{region '#Template'}
	{attribute 'Version' := '5.0.1.0'}
	{attribute 'Tags' := '"LCID": "1031", "Text": "Universal, Motor, Aggregate"'}
	{attribute 'Tags' := '"LCID": "1033", "Text": "Universal, Motor, Aggregate"'}
	{attribute 'Using' := '"Type": "Template", "URI": "EC_ID"'}
	{attribute 'Using' := '"Type": "Template", "URI": "BA2_Param"'}
	{attribute 'Description' := '"LCID": "1031", "Text": "Motor modulierend mit Regler"'}
	{attribute 'Description' := '"LCID": "1033", "Text": "Motor modulating with controller"'}
{endregion}		
FUNCTION_BLOCK FB_BA_MotCtl EXTENDS FB_BA_View
VAR_INPUT
	fIn				: REAL;	// Istwert Regler // Actual value controller	
	stCmd			: ST_BA_Mdlt;
END_VAR
VAR_OUTPUT
	bCmd			: BOOL;
	fMdlt			: REAL;
	bDst			: BOOL;
	eActivePrio		: E_BA_Priority;
END_VAR

VAR_INPUT CONSTANT
	Dst				: FB_BA_BI_Raw;
	Cmd				: FB_BA_BO_Raw;								 
	Mdlt			: FB_BA_AO_Raw;							
	Sp				: FB_BA_AV_Op;		 
	Ctrl			: FB_BA_Loop;		
	PlantLock		: FB_BA_PlantLock;														
END_VAR
VAR
	bPrioSfty					: BOOL;
	bPrioCrit					: BOOL;	
	
	PrioSwiVal					: FB_BA_PrioSwi_UDI04;	

	MuxCmd						: FB_BA_MMUX_B04;
	MuxMdlt						: FB_BA_MMUX_R04;
	fMax						: REAL;
	fMin						: REAL;		
END_VAR
VAR // added by the converter: edge detectors and wires of the graphical bodies
    _w1, _w2 : ANY;
END_VAR

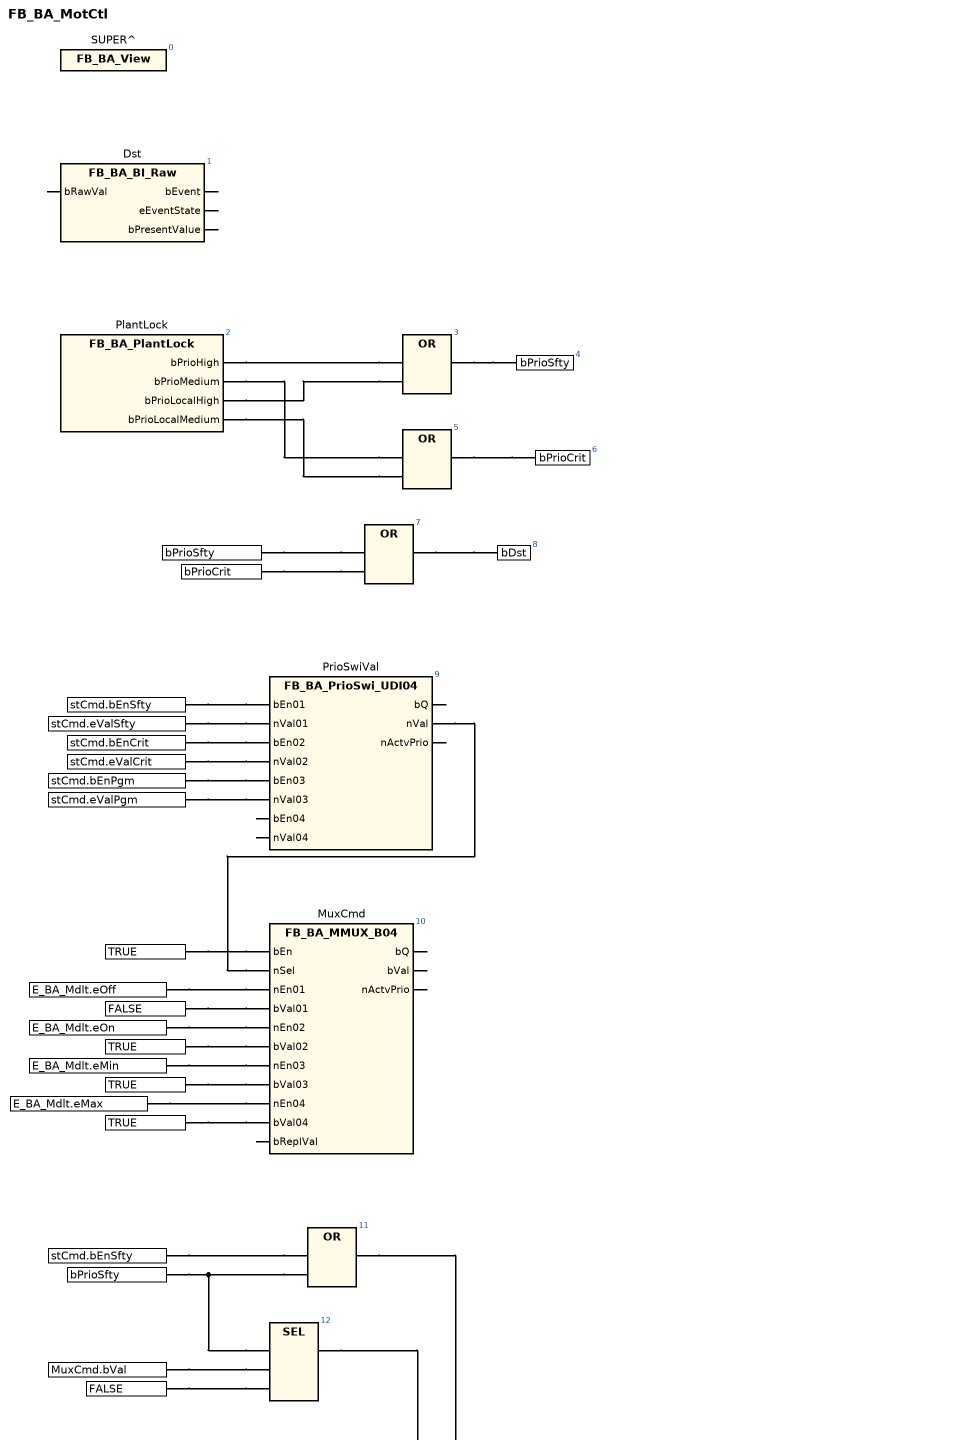
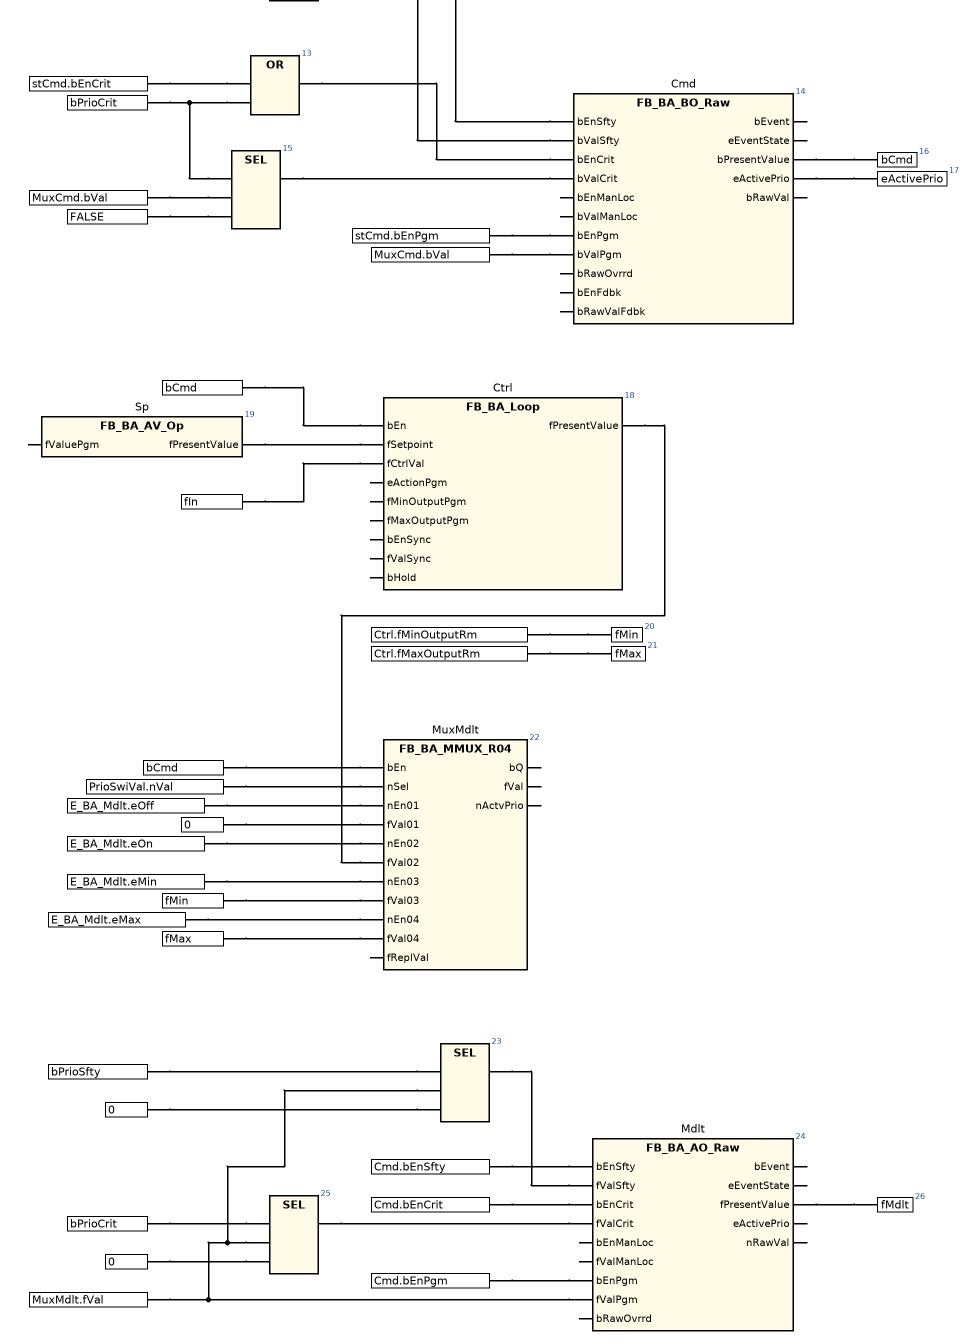
SUPER^(); // FB_BA_View
Dst(); // FB_BA_BI_Raw
PlantLock(); // FB_BA_PlantLock
bPrioSfty := PlantLock.bPrioHigh OR PlantLock.bPrioLocalHigh;
bPrioCrit := PlantLock.bPrioMedium OR PlantLock.bPrioLocalMedium;
bDst := bPrioSfty OR bPrioCrit;
PrioSwiVal(
    bEn01 := stCmd.bEnSfty,
    nVal01 := stCmd.eValSfty,
    bEn02 := stCmd.bEnCrit,
    nVal02 := stCmd.eValCrit,
    bEn03 := stCmd.bEnPgm,
    nVal03 := stCmd.eValPgm); // FB_BA_PrioSwi_UDI04
MuxCmd(
    bEn := TRUE,
    nSel := PrioSwiVal.nVal,
    nEn01 := E_BA_Mdlt.eOff,
    bVal01 := FALSE,
    nEn02 := E_BA_Mdlt.eOn,
    bVal02 := TRUE,
    nEn03 := E_BA_Mdlt.eMin,
    bVal03 := TRUE,
    nEn04 := E_BA_Mdlt.eMax,
    bVal04 := TRUE); // FB_BA_MMUX_B04
Cmd(
    bEnSfty := stCmd.bEnSfty OR bPrioSfty,
    bValSfty := SEL(bPrioSfty, MuxCmd.bVal, FALSE),
    bEnCrit := stCmd.bEnCrit OR bPrioCrit,
    bValCrit := _w1,
    bEnPgm := stCmd.bEnPgm,
    bValPgm := MuxCmd.bVal); // FB_BA_BO_Raw
_w1 := SEL(bPrioCrit, MuxCmd.bVal, FALSE);
bCmd := Cmd.bPresentValue;
eActivePrio := Cmd.eActivePrio;
Ctrl(bEn := bCmd, fSetpoint := Sp.fPresentValue, fCtrlVal := fIn); // FB_BA_Loop
Sp(); // FB_BA_AV_Op
fMin := Ctrl.fMinOutputRm;
fMax := Ctrl.fMaxOutputRm;
MuxMdlt(
    bEn := bCmd,
    nSel := PrioSwiVal.nVal,
    nEn01 := E_BA_Mdlt.eOff,
    fVal01 := 0,
    nEn02 := E_BA_Mdlt.eOn,
    fVal02 := Ctrl.fPresentValue,
    nEn03 := E_BA_Mdlt.eMin,
    fVal03 := fMin,
    nEn04 := E_BA_Mdlt.eMax,
    fVal04 := fMax); // FB_BA_MMUX_R04
Mdlt(
    bEnSfty := Cmd.bEnSfty,
    fValSfty := SEL(bPrioSfty, MuxMdlt.fVal, 0),
    bEnCrit := Cmd.bEnCrit,
    fValCrit := _w2,
    bEnPgm := Cmd.bEnPgm,
    fValPgm := MuxMdlt.fVal); // FB_BA_AO_Raw
_w2 := SEL(bPrioCrit, MuxMdlt.fVal, 0);
fMdlt := Mdlt.fPresentValue;

METHOD FB_init : BOOL
VAR_INPUT
	bInitRetains : BOOL; // if TRUE, the retain variables are initialized (warm start / cold start)
	bInCopyCode : BOOL;  // if TRUE, the instance afterwards gets moved into the copy code (online change)
END_VAR
PlantLock.Parent					:= THIS^;		

Dst.iParent							:= THIS^;
Dst.iLabel							:= LblFun_Fault;  
Dst.ePolarity						:= E_BA_Polarity.eReverse;
Dst.sActiveText 					:= txtEvent_Triggered;
Dst.sInactiveText 					:= txtEvent_Normal;
Dst.nEventClassID					:= EC_ID.NC30;
Dst.stTimeDelay.nToNormal			:= BA2_Param.nDefTimeDelay_ToNormal;
Dst.stTimeDelay.nToAbnormal			:= BA2_Param.nDefTimeDelay_ToAbnormal;
Dst.bAlarmValue						:= TRUE;
Dst.aEventTransitionText[1]			:= txtEvent_Triggered;
Dst.aEventTransitionText[2]			:= txtEvent_Error;
Dst.aEventTransitionText[3]			:= txtEvent_Normal;
Dst.bEventDetectionEnable			:= TRUE;
Dst.eEnPlantLock					:= E_BA_LockPriority.eLocalMedium;

Cmd.iParent							:= THIS^;
Cmd.iLabel							:= LblFun_SwitchingCommand;  
Cmd.ePolarity						:= E_BA_Polarity.eNormal;
Cmd.sActiveText 					:= txtEvent_On;
Cmd.sInactiveText 					:= txtEvent_Off;
Cmd.bEnManualRm						:= FALSE;	//	Priority  8	
Cmd.bValManualRm					:= FALSE;	//	Priority  8
Cmd.nEventClassID					:= EC_ID.NC40;
Cmd.stTimeDelay.nToNormal			:= BA2_Param.nDefTimeDelay_ToNormal;
Cmd.stTimeDelay.nToAbnormal			:= BA2_Param.nDefTimeDelay_ToAbnormal;
Cmd.aEventTransitionText[1]			:= txtEvent_Disturb;
Cmd.aEventTransitionText[2]			:= txtEvent_None;
Cmd.aEventTransitionText[3]			:= txtEvent_Normal;
Cmd.bEventDetectionEnable			:= FALSE;
Cmd.eEnPlantLock					:= E_BA_LockPriority.eNoLock;

Mdlt.iParent						:= THIS^;
Mdlt.iLabel							:= LblFun_ControlSignal;  
Mdlt.eUnit							:= E_BA_Unit.eOther_Percent;
Mdlt.fResolution 					:= 0.003051851;
Mdlt.fScaleOffset 					:= 0;
Mdlt.fCOVIncrement					:= BA2_Param.fDefCOVIncrement;
Mdlt.bEnManualRm					:= FALSE;	//	Priority  8	
Mdlt.fValManualRm					:= 0.0;		//	Priority  8
Mdlt.nEventClassID					:= EC_ID.NC80;
Mdlt.stTimeDelay.nToNormal			:= BA2_Param.nDefTimeDelay_ToNormal;
Mdlt.stTimeDelay.nToAbnormal		:= BA2_Param.nDefTimeDelay_ToAbnormal;
Mdlt.stHighLimit.bEnable			:= FALSE;
Mdlt.stHighLimit.fValue				:= 0.0;		
Mdlt.stLowLimit.bEnable				:= FALSE;
Mdlt.stLowLimit.fValue				:= 0.0;
Mdlt.fLimitDeadband 				:= BA2_Param.fDefLimitDeadband;
Mdlt.aEventTransitionText[1]		:= txtEvent_Disturb;
Mdlt.aEventTransitionText[2]		:= txtEvent_None;
Mdlt.aEventTransitionText[3]		:= txtEvent_Normal;
Mdlt.bEventDetectionEnable			:= FALSE;
Mdlt.eEnPlantLock					:= E_BA_LockPriority.eNoLock;

Sp.iParent							:= THIS^;
Sp.iLabel							:= LblFun_Setpoint; 
Sp.eUnit 							:= E_BA_Unit.ePressure_Pascals;								 
Sp.fValueRm							:= 250;
Sp.fCOVIncrement					:= BA2_Param.fDefCOVIncrement;

Ctrl.iParent						:= THIS^;
Ctrl.iLabel							:= LblFun_LoopObject;  
Ctrl.eOpMode						:= E_BA_PIDMode.ePID;								 	 										 
Ctrl.eOutputUnit					:= E_BA_Unit.eOther_Percent;
Ctrl.eActionRm						:= E_BA_Action.eReverse;
Ctrl.fProportionalConstant			:= 0.01;
Ctrl.fIntegralConstant				:= 60;
Ctrl.fDerivativeConstant			:= 0;
Ctrl.fMaxOutputRm 					:= 100;
Ctrl.fMinOutputRm					:= 20;
Ctrl.fCOVIncrement					:= 0;
Ctrl.nDampConstant					:= 0;
Ctrl.fNeutralZone					:= 0;
END_METHOD

END_FUNCTION_BLOCK

(* stored: Version 1.1.0.1, ProductVersion 3.1.4024.15
   POU FB_BA_MotCtl: Id {e9537c15-7884-45d0-b4c9-e74be163c3d6}, SpecialFunc None
   Method FB_init: Id {f6450f97-f524-4df9-ab99-bd2a799100fd} *)
